Staubli VAL3: default.pjx

Parameters millimeterUnit=true stackSize=5000 version=s8.12.3cs9_BS2740
Program file=start.pgx
Program file=stop.pgx
Data file=default.dtx
